Universal Robots URScript: rubik.script

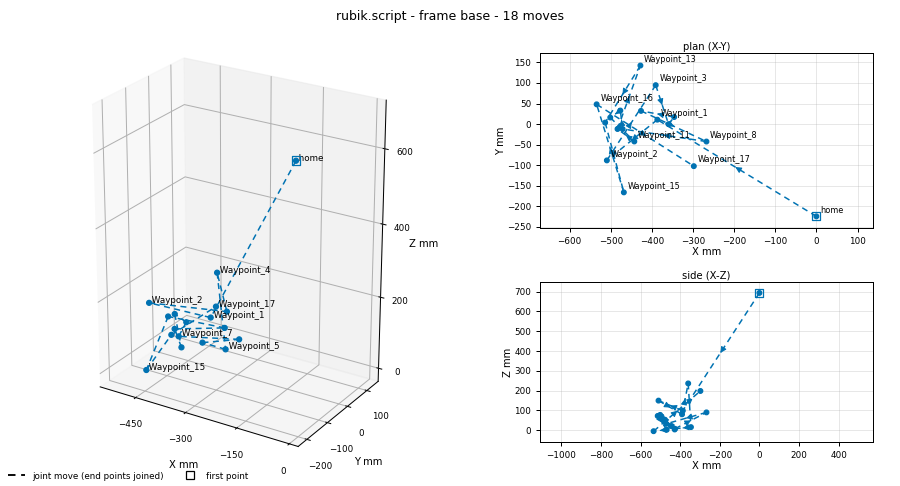
[picture p0: tool path of rubik.script in frame base, 18 of 18 moves have a stored position in this frame; points joined in program order, loops and branches not executed]
def unnamed():
  global _hidden_verificationVariable=0
  set_safety_mode_transition_hardness(1)
  set_standard_analog_input_domain(0, 1)
  set_standard_analog_input_domain(1, 1)
  set_tool_analog_input_domain(0, 1)
  set_tool_analog_input_domain(1, 1)
  set_analog_outputdomain(0, 0)
  set_analog_outputdomain(1, 0)
  set_input_actions_to_default()
  set_target_payload(0.050000, [0.000000, 0.000000, 0.000000], [0.000010, 0.000010, 0.000010, 0.000000, 0.000000, 0.000000])
  set_tcp(p[0.0,0.0,0.0,0.0,0.0,0.0])
  set_tool_communication(False, 115200, 0, 1, 1.5, 3.5)
  set_tool_output_mode(0)
  set_tool_digital_output_mode(0, 1)
  set_tool_digital_output_mode(1, 1)
  set_tool_voltage(0)
  modbus_add_signal("192.168.1.101", 255, 0, 2, "MODBUS_1", False)
  modbus_set_signal_update_frequency("MODBUS_1", 10)
  modbus_add_signal("192.168.1.101", 255, 0, 2, "MODBUS_2", False)
  modbus_set_signal_update_frequency("MODBUS_2", 10)
  set_gravity([0.0, 0.0, 9.82])
  step_count_388f09be_3944_469c_8391_754207b1bb49 = 0.0
  thread Step_Counter_Thread_7694d8d0_05e8_4a58_82d1_653fb5794752():
    while (True):
      step_count_388f09be_3944_469c_8391_754207b1bb49 = step_count_388f09be_3944_469c_8391_754207b1bb49 + 1.0
      sync()
    end
  end
  run Step_Counter_Thread_7694d8d0_05e8_4a58_82d1_653fb5794752()
  global home_p=p[-.000275677407, -.224354758206, .693295766768, -.000588461133, -2.227685077545, 2.214755080677]
  global home_q=[3.254189869039692E-5, -1.5707877227744866, -1.1435984561103396E-5, -1.5707760242279, -2.9865895406544496E-5, 3.3714073651935905E-5]
  global Waypoint_1_p=p[-.386953497294, .010673819392, .098882036830, -2.361225367261, -1.835428132246, .588231554425]
  global Waypoint_1_q=[-0.45118695894350225, -0.9367697995952149, 2.002096954976217, -2.903895994225973, -1.269067112599508, -0.1577680746661585]
  global Waypoint_2_p=p[-.509655359247, -.088307579985, .149724556371, -2.139818610402, -1.239595347355, -.513365052047]
  global Waypoint_2_q=[0.03541717678308487, -0.43431885660205083, 0.5746548811541956, -1.6399270496764125, -2.302408997212545, 0.5858011245727539]
  global Waypoint_3_p=p[-.390858657819, .094615060967, .080557865089, 2.382204565498, 1.419939914968, -.914877027991]
  global Waypoint_3_q=[-0.7271969954120081, -0.8578885954669495, 1.8743379751788538, -2.56481470684194, -0.8980420271502894, -0.23550159135927373]
  global Waypoint_4_p=p[-.359767779282, -.000224843325, .236477994854, -2.173373684142, -1.860482926068, .338858193912]
  global Waypoint_4_q=[-0.3995454947101038, -1.4422534567168732, 1.9229524771319788, -2.393491407433981, -1.4791458288775843, -0.225626293812887]
  global Waypoint_5_p=p[-.345973112813, .017074143962, .015890143730, 2.059361185402, 1.747226794813, .270453686389]
  global Waypoint_5_q=[-0.4389446417437952, -0.7605455678752442, 1.7908762137042444, -2.1323067150511683, -1.570641819630758, -0.2722380797015589]
  global Waypoint_6_p=p[-.426655153210, .032033957376, .007582810082, 2.323987682208, 2.015638039561, -.095786347416]
  global Waypoint_6_q=[-0.40693599382509404, -0.5601480764201661, 1.55792743364443, -2.540586610833639, -1.4875128904925745, -0.2630246321307581]
  global Waypoint_8_p=p[-.267550828096, -.042468190649, .090262075370, -2.185200546977, -1.737572770756, .500881268059]
  global Waypoint_8_q=[-0.4127414862262171, -0.9275530141643067, 2.6582608858691614, -3.7437812290587367, -1.4099515120135706, -0.14773160616029912]
  global Waypoint_7_p=p[-.471288661788, -.011994513971, .032512518962, 2.631078792328, 1.502906786262, .136748896998]
  global Waypoint_7_q=[-0.26081639925111944, -0.5001546901515503, 1.1723998228656214, -2.1049701176085414, -1.5564811865436, 0.27442440390586853]
  global Waypoint_9_p=p[-.476885745483, .032879088445, .053244743282, 2.519393628375, 1.141554183822, -.292051642577]
  global Waypoint_9_q=[-0.42613107362856084, -0.5559906524470826, 1.2163713614093226, -2.093163629571432, -1.17702562013735, 0.2700496315956116]
  global Waypoint_10_p=p[-.501365756117, .015925567065, .077659939913, 2.632740013057, 1.423202495600, -.286296572546]
  global Waypoint_10_q=[-0.3419235388385218, -0.5420174163630982, 1.0974019209491175, -2.1567098102965296, -1.3384316603290003, 0.24497056007385254]
  global Waypoint_11_p=p[-.442898092933, -.042282244367, .021054898242, -2.082485528954, -1.688860918050, -.918947397981]
  global Waypoint_11_q=[-0.07358438173402959, -0.4483298820308228, 1.1708410421954554, -1.9828278026976527, -2.237105194722311, 0.24524393677711487]
  global Waypoint_12_p=p[-.483715305322, -.011954488137, .050710788045, -2.235072925205, -1.530246968621, -.593597678816]
  global Waypoint_12_q=[-0.14708120027651006, -0.4367574018291016, 1.0359228293048304, -2.102835317651266, -2.13235313097109, 0.24515067040920258]
  global Waypoint_13_p=p[-.428054704570, .142338687149, .003997808408, 2.640162754677, 1.642870468547, .010281221286]
  global Waypoint_13_q=[-0.6188133398639124, -0.48485787332568364, 1.3799894491778772, -2.4361125431456507, -1.5649169127093714, -0.15812188783754522]
  global Waypoint_14_p=p[-.513761591350, .003590199789, .072415117663, -2.231328553260, -1.990574526804, .373305082922]
  global Waypoint_14_q=[-0.2931450049029749, -0.4860835832408448, 1.1117046515094202, -2.439934392968649, -1.4284070173846644, -0.15817767778505498]
  global Waypoint_15_p=p[-.468371893520, -.166051046455, .002615356969, 2.157492554948, 2.164246139214, -.074794099199]
  global Waypoint_15_q=[0.053705181926488876, -0.34017785013232427, 1.0373767058001917, -2.2501231632628382, -1.4752123991595667, 0.053198203444480896]
  global Waypoint_16_p=p[-.534522367155, .048005648038, -.004715374303, -2.290802083289, -2.050208240438, .204328388447]
  global Waypoint_16_q=[-0.35357982317079717, -0.14992590368304448, 0.7001951376544397, -2.2395688496031703, -1.4826024214373987, -0.2341559568988245]
  global Waypoint_17_p=p[-.298201406555, -.102335740089, .198335331537, -1.513456321991, -1.630209929433, .355833618723]
  global Waypoint_17_q=[0.007939094677567482, -1.2048554581454773, 2.335468594227926, -3.596079488793844, -1.9211228529559534, -0.23344546953310186]
  $ 1 "Robot Program"
  $ 2 "MoveJ"
  $ 3 "home" "breakAfter"
  movej(get_inverse_kin(home_p, qnear=home_q), a=6.283185307179586, v=6.283185307179586)
  $ 4 "MoveJ"
  $ 5 "Waypoint_1" "breakAfter"
  movej(get_inverse_kin(Waypoint_1_p, qnear=Waypoint_1_q), a=6.1086523819801535, v=6.1086523819801535)
  $ 6 "Waypoint_2" "breakAfter"
  movej(get_inverse_kin(Waypoint_2_p, qnear=Waypoint_2_q), a=2.6179938779914944, v=3.490658503988659)
  $ 7 "Wait: 0.3"
  sleep(0.3)
  $ 8 "Waypoint_3" "breakAfter"
  movej(get_inverse_kin(Waypoint_3_p, qnear=Waypoint_3_q), a=1.3962634015954636, v=3.490658503988659)
  $ 9 "Wait: 0.5"
  sleep(0.5)
  $ 10 "Waypoint_4" "breakAfter"
  movej(get_inverse_kin(Waypoint_4_p, qnear=Waypoint_4_q), a=1.3962634015954636, v=2.6179938779914944)
  $ 11 "Waypoint_5" "breakAfter"
  movej(get_inverse_kin(Waypoint_5_p, qnear=Waypoint_5_q), a=0.8726646259971648, v=0.8726646259971648)
  $ 12 "Waypoint_6" "breakAfter"
  movej(get_inverse_kin(Waypoint_6_p, qnear=Waypoint_6_q), a=6.1086523819801535, v=6.1086523819801535)
  $ 13 "Waypoint_8" "breakAfter"
  movej(get_inverse_kin(Waypoint_8_p, qnear=Waypoint_8_q), a=6.1086523819801535, v=6.1086523819801535)
  $ 14 "Wait: 1.0"
  sleep(1.0)
  $ 15 "Waypoint_7" "breakAfter"
  movej(get_inverse_kin(Waypoint_7_p, qnear=Waypoint_7_q), a=1.3962634015954636, v=1.0471975511965976)
  $ 16 "Waypoint_9" "breakAfter"
  movej(get_inverse_kin(Waypoint_9_p, qnear=Waypoint_9_q), a=6.1086523819801535, v=6.1086523819801535)
  $ 17 "Waypoint_10" "breakAfter"
  movej(get_inverse_kin(Waypoint_10_p, qnear=Waypoint_10_q), a=6.1086523819801535, v=6.1086523819801535)
  $ 18 "Waypoint_11" "breakAfter"
  movej(get_inverse_kin(Waypoint_11_p, qnear=Waypoint_11_q), a=6.1086523819801535, v=6.1086523819801535)
  $ 19 "Waypoint_12" "breakAfter"
  movej(get_inverse_kin(Waypoint_12_p, qnear=Waypoint_12_q), a=6.1086523819801535, v=6.1086523819801535)
  $ 20 "Waypoint_13" "breakAfter"
  movej(get_inverse_kin(Waypoint_13_p, qnear=Waypoint_13_q), a=6.1086523819801535, v=6.1086523819801535)
  $ 21 "Waypoint_14" "breakAfter"
  movej(get_inverse_kin(Waypoint_14_p, qnear=Waypoint_14_q), a=6.1086523819801535, v=6.1086523819801535)
  $ 22 "Waypoint_15" "breakAfter"
  movej(get_inverse_kin(Waypoint_15_p, qnear=Waypoint_15_q), a=6.1086523819801535, v=6.1086523819801535)
  $ 23 "Waypoint_16" "breakAfter"
  movej(get_inverse_kin(Waypoint_16_p, qnear=Waypoint_16_q), a=6.1086523819801535, v=6.1086523819801535)
  $ 24 "Waypoint_17" "breakAfter"
  movej(get_inverse_kin(Waypoint_17_p, qnear=Waypoint_17_q), a=6.1086523819801535, v=6.1086523819801535)
end
